(* Logix 5000 project; controller Amvex_Thorpe_Flowmeter vendor 1 type 14 code 106 rev 33.13; software revision 33.01; part 4 of 16 *)

ADD_ON_INSTRUCTION MoveLinRelTRF   (* revision 0.1, vendor Mecademic Inc., ExecuteEnableInFalse *)
// Relative movement (relative to the current TRF position)
VAR_IN_OUT
   RobotInputs : _061D:Meca500_86BDA20B:I:0; {required}
   RobotOutputs : _061D:Meca500_01F88326:O:0; {required}
END_VAR
VAR_INPUT
   Pose_X_Pos : REAL; {required}
   Pose_Y_Pos : REAL; {required}
   Pose_Z_Pos : REAL; {required}
   Pose_rX_Ang : REAL; {required}
   Pose_rY_Ang : REAL; {required}
   Pose_rZ_Ang : REAL; {required}
   ExternalStateControl : BOOL; {required}
   ExternalMoveID : INT; {required}
END_VAR
VAR_OUTPUT
   Enabled : BOOL; {visible}
   Sent : BOOL; {visible}
   Buffered : BOOL; {visible}
   Error : BOOL; {visible}
END_VAR
VAR
   InternalMoveID : INT; {access None}
   MoveIDTrig : BOOL; {access None}
   MoveIDUpdated : BOOL; {access None}
   OneShot : DINT; {access None}
   FirstScan : BOOL; {access None}
END_VAR

ROUTINE EnableInFalse   (* ladder *)
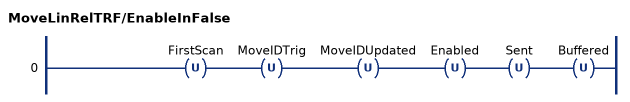
   0: OTU(FirstScan)OTU(MoveIDTrig)OTU(MoveIDUpdated)OTU(Enabled)OTU(Sent)OTU(Buffered);
END_ROUTINE

ROUTINE Logic   (* ladder *)
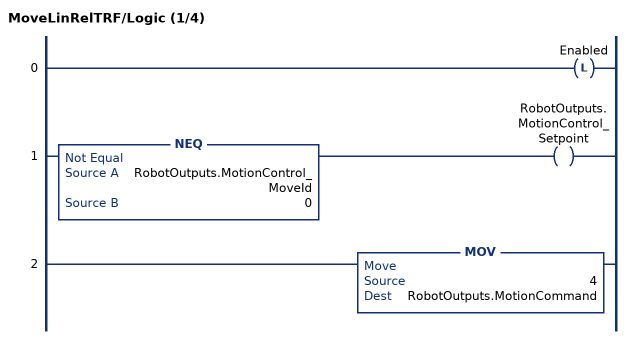
   0: OTL(Enabled);
   1: NEQ(RobotOutputs.MotionControl_MoveId,0)OTE(RobotOutputs.MotionControl_Setpoint);
   2: MOV(4,RobotOutputs.MotionCommand);
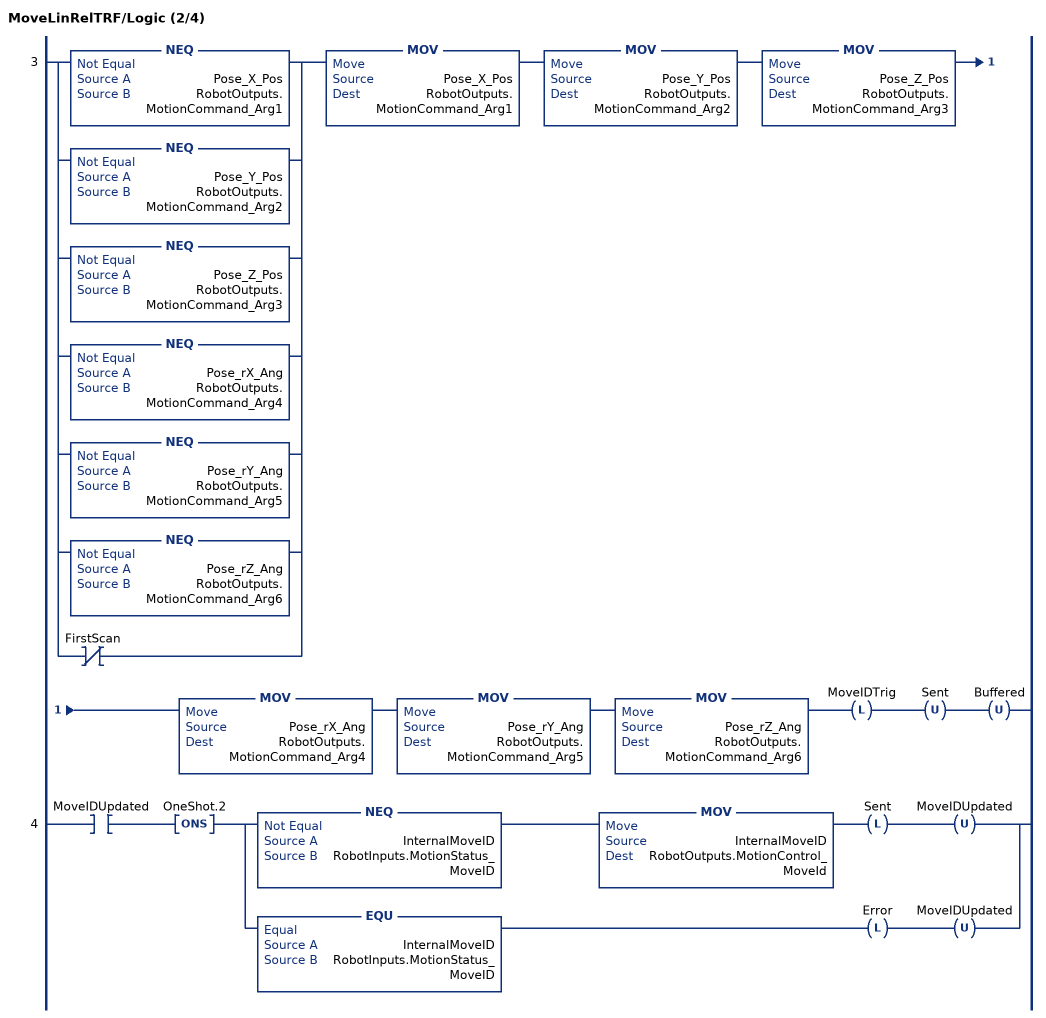
   3: [NEQ(Pose_X_Pos,RobotOutputs.MotionCommand_Arg1) ,NEQ(Pose_Y_Pos,RobotOutputs.MotionCommand_Arg2) ,NEQ(Pose_Z_Pos,RobotOutputs.MotionCommand_Arg3) ,NEQ(Pose_rX_Ang,RobotOutputs.MotionCommand_Arg4) ,NEQ(Pose_rY_Ang,RobotOutputs.MotionCommand_Arg5) ,NEQ(Pose_rZ_Ang,RobotOutputs.MotionCommand_Arg6) ,XIO(FirstScan) ]MOV(Pose_X_Pos,RobotOutputs.MotionCommand_Arg1)MOV(Pose_Y_Pos,RobotOutputs.MotionCommand_Arg2)MOV(Pose_Z_Pos,RobotOutputs.MotionCommand_Arg3)MOV(Pose_rX_Ang,RobotOutputs.MotionCommand_Arg4)MOV(Pose_rY_Ang,RobotOutputs.MotionCommand_Arg5)MOV(Pose_rZ_Ang,RobotOutputs.MotionCommand_Arg6)OTL(MoveIDTrig)OTU(Sent)OTU(Buffered);
   4: XIC(MoveIDUpdated)ONS(OneShot.2)[NEQ(InternalMoveID,RobotInputs.MotionStatus_MoveID) MOV(InternalMoveID,RobotOutputs.MotionControl_MoveId) OTL(Sent) OTU(MoveIDUpdated) ,EQU(InternalMoveID,RobotInputs.MotionStatus_MoveID) OTL(Error) OTU(MoveIDUpdated) ];
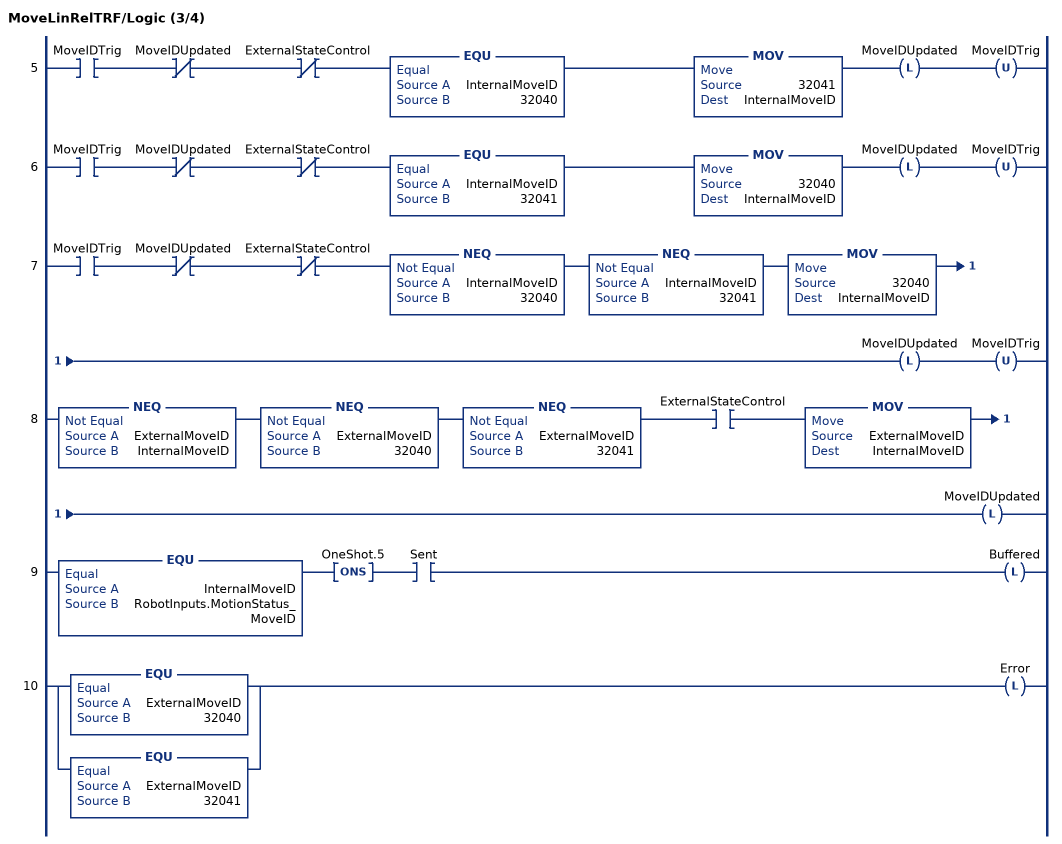
   5: XIC(MoveIDTrig)XIO(MoveIDUpdated)XIO(ExternalStateControl)EQU(InternalMoveID,32040)MOV(32041,InternalMoveID)OTL(MoveIDUpdated)OTU(MoveIDTrig);
   6: XIC(MoveIDTrig)XIO(MoveIDUpdated)XIO(ExternalStateControl)EQU(InternalMoveID,32041)MOV(32040,InternalMoveID)OTL(MoveIDUpdated)OTU(MoveIDTrig);
   7: XIC(MoveIDTrig)XIO(MoveIDUpdated)XIO(ExternalStateControl)NEQ(InternalMoveID,32040)NEQ(InternalMoveID,32041)MOV(32040,InternalMoveID)OTL(MoveIDUpdated)OTU(MoveIDTrig);
   8: NEQ(ExternalMoveID,InternalMoveID)NEQ(ExternalMoveID,32040)NEQ(ExternalMoveID,32041)XIC(ExternalStateControl)MOV(ExternalMoveID,InternalMoveID)OTL(MoveIDUpdated);
   9: EQU(InternalMoveID,RobotInputs.MotionStatus_MoveID)ONS(OneShot.5)XIC(Sent)OTL(Buffered);
   10: [EQU(ExternalMoveID,32040) ,EQU(ExternalMoveID,32041) ]OTL(Error);
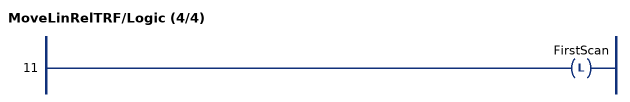
   11: OTL(FirstScan);
END_ROUTINE
END_ADD_ON_INSTRUCTION

ADD_ON_INSTRUCTION MoveLinRelWRF   (* revision 0.1, vendor Mecademic Inc., ExecuteEnableInFalse *)
// Relative movement (relative to the current WRF position)
VAR_IN_OUT
   RobotInputs : _061D:Meca500_86BDA20B:I:0; {required}
   RobotOutputs : _061D:Meca500_01F88326:O:0; {required}
END_VAR
VAR_INPUT
   Pose_X_Pos : REAL; {required}
   Pose_Y_Pos : REAL; {required}
   Pose_Z_Pos : REAL; {required}
   Pose_rX_Ang : REAL; {required}
   Pose_rY_Ang : REAL; {required}
   Pose_rZ_Ang : REAL; {required}
   ExternalStateControl : BOOL; {required}
   ExternalMoveID : INT; {required}
END_VAR
VAR_OUTPUT
   Enabled : BOOL; {visible}
   Sent : BOOL; {visible}
   Buffered : BOOL; {visible}
   Error : BOOL; {visible}
END_VAR
VAR
   InternalMoveID : INT; {access None}
   MoveIDTrig : BOOL; {access None}
   MoveIDUpdated : BOOL; {access None}
   OneShot : DINT; {access None}
   FirstScan : BOOL; {access None}
END_VAR

ROUTINE EnableInFalse   (* ladder *)
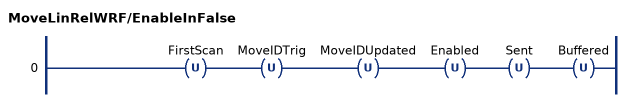
   0: OTU(FirstScan)OTU(MoveIDTrig)OTU(MoveIDUpdated)OTU(Enabled)OTU(Sent)OTU(Buffered);
END_ROUTINE

ROUTINE Logic   (* ladder *)
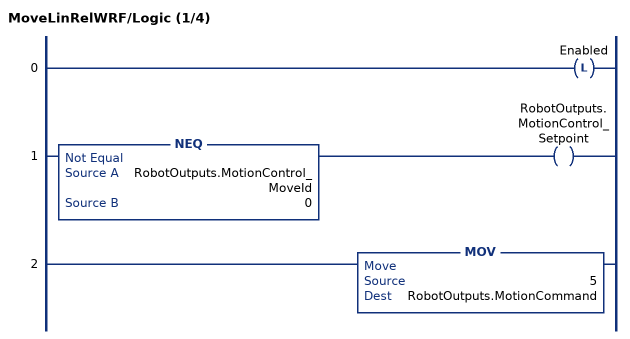
   0: OTL(Enabled);
   1: NEQ(RobotOutputs.MotionControl_MoveId,0)OTE(RobotOutputs.MotionControl_Setpoint);
   2: MOV(5,RobotOutputs.MotionCommand);
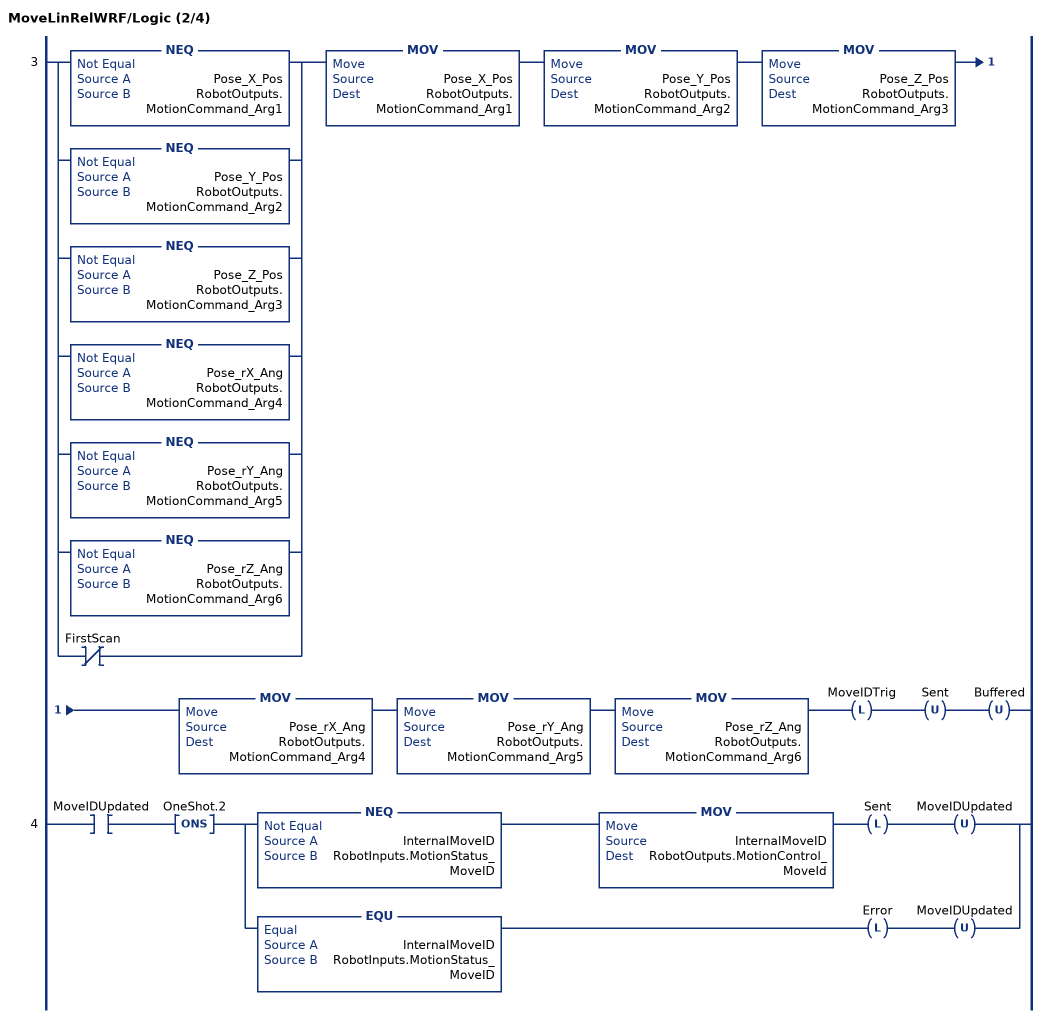
   3: [NEQ(Pose_X_Pos,RobotOutputs.MotionCommand_Arg1) ,NEQ(Pose_Y_Pos,RobotOutputs.MotionCommand_Arg2) ,NEQ(Pose_Z_Pos,RobotOutputs.MotionCommand_Arg3) ,NEQ(Pose_rX_Ang,RobotOutputs.MotionCommand_Arg4) ,NEQ(Pose_rY_Ang,RobotOutputs.MotionCommand_Arg5) ,NEQ(Pose_rZ_Ang,RobotOutputs.MotionCommand_Arg6) ,XIO(FirstScan) ]MOV(Pose_X_Pos,RobotOutputs.MotionCommand_Arg1)MOV(Pose_Y_Pos,RobotOutputs.MotionCommand_Arg2)MOV(Pose_Z_Pos,RobotOutputs.MotionCommand_Arg3)MOV(Pose_rX_Ang,RobotOutputs.MotionCommand_Arg4)MOV(Pose_rY_Ang,RobotOutputs.MotionCommand_Arg5)MOV(Pose_rZ_Ang,RobotOutputs.MotionCommand_Arg6)OTL(MoveIDTrig)OTU(Sent)OTU(Buffered);
   4: XIC(MoveIDUpdated)ONS(OneShot.2)[NEQ(InternalMoveID,RobotInputs.MotionStatus_MoveID) MOV(InternalMoveID,RobotOutputs.MotionControl_MoveId) OTL(Sent) OTU(MoveIDUpdated) ,EQU(InternalMoveID,RobotInputs.MotionStatus_MoveID) OTL(Error) OTU(MoveIDUpdated) ];
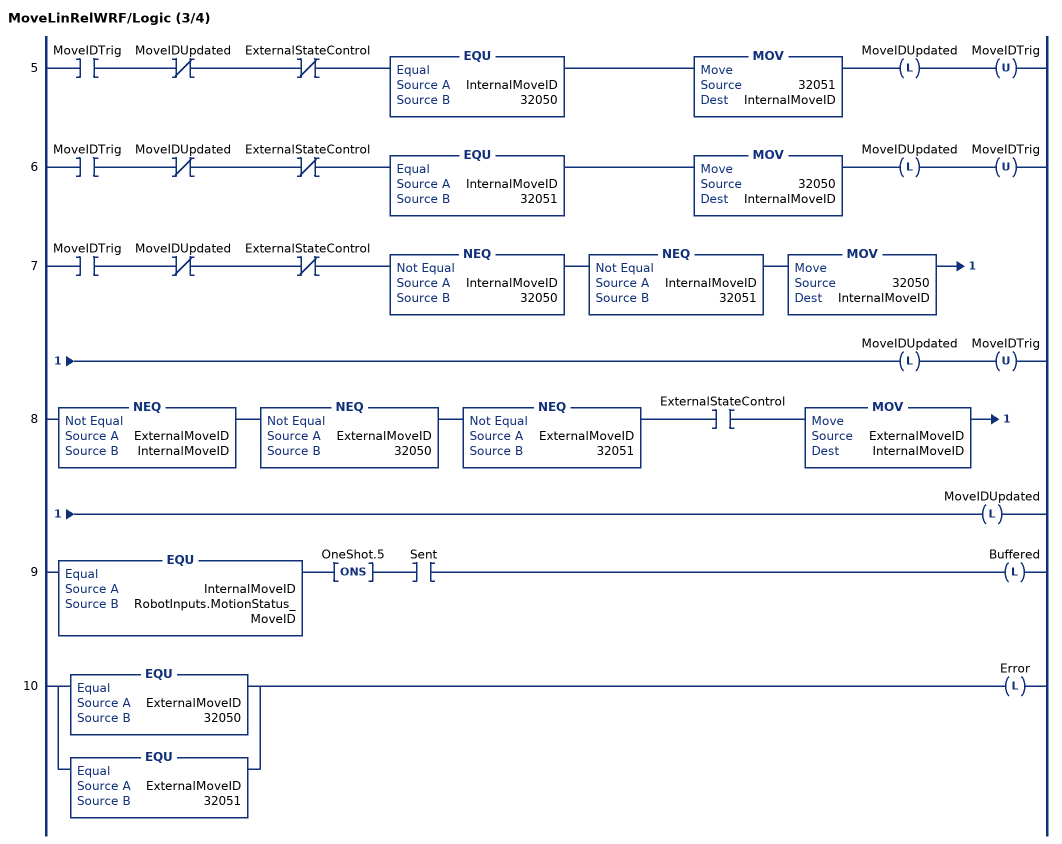
   5: XIC(MoveIDTrig)XIO(MoveIDUpdated)XIO(ExternalStateControl)EQU(InternalMoveID,32050)MOV(32051,InternalMoveID)OTL(MoveIDUpdated)OTU(MoveIDTrig);
   6: XIC(MoveIDTrig)XIO(MoveIDUpdated)XIO(ExternalStateControl)EQU(InternalMoveID,32051)MOV(32050,InternalMoveID)OTL(MoveIDUpdated)OTU(MoveIDTrig);
   7: XIC(MoveIDTrig)XIO(MoveIDUpdated)XIO(ExternalStateControl)NEQ(InternalMoveID,32050)NEQ(InternalMoveID,32051)MOV(32050,InternalMoveID)OTL(MoveIDUpdated)OTU(MoveIDTrig);
   8: NEQ(ExternalMoveID,InternalMoveID)NEQ(ExternalMoveID,32050)NEQ(ExternalMoveID,32051)XIC(ExternalStateControl)MOV(ExternalMoveID,InternalMoveID)OTL(MoveIDUpdated);
   9: EQU(InternalMoveID,RobotInputs.MotionStatus_MoveID)ONS(OneShot.5)XIC(Sent)OTL(Buffered);
   10: [EQU(ExternalMoveID,32050) ,EQU(ExternalMoveID,32051) ]OTL(Error);
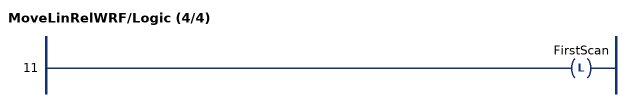
   11: OTL(FirstScan);
END_ROUTINE
END_ADD_ON_INSTRUCTION

ADD_ON_INSTRUCTION MoveLinVelTRF   (* revision 0.1, vendor Mecademic Inc., ExecuteEnableInFalse *)
// Set current mode to "cartesian TRF velocity mode"
VAR_IN_OUT
   RobotInputs : _061D:Meca500_86BDA20B:I:0; {required}
   RobotOutputs : _061D:Meca500_01F88326:O:0; {required}
END_VAR
VAR_INPUT
   Pose_X_Vel : REAL; {required}
   Pose_Y_Vel : REAL; {required}
   Pose_Z_Vel : REAL; {required}
   Pose_rX_Vel : REAL; {required}
   Pose_rY_Vel : REAL; {required}
   Pose_rZ_Vel : REAL; {required}
   ExternalStateControl : BOOL; {required}
   ExternalMoveID : INT; {required}
END_VAR
VAR_OUTPUT
   Enabled : BOOL; {visible}
   Sent : BOOL; {visible}
   Buffered : BOOL; {visible}
   Error : BOOL; {visible}
END_VAR
VAR
   InternalMoveID : INT; {access None}
   MoveIDTrig : BOOL; {access None}
   MoveIDUpdated : BOOL; {access None}
   OneShot : DINT; {access None}
   FirstScan : BOOL; {access None}
END_VAR

ROUTINE EnableInFalse   (* ladder *)
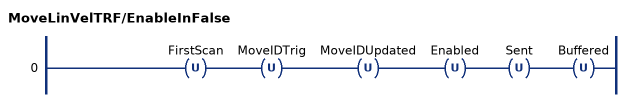
   0: OTU(FirstScan)OTU(MoveIDTrig)OTU(MoveIDUpdated)OTU(Enabled)OTU(Sent)OTU(Buffered);
END_ROUTINE

ROUTINE Logic   (* ladder *)
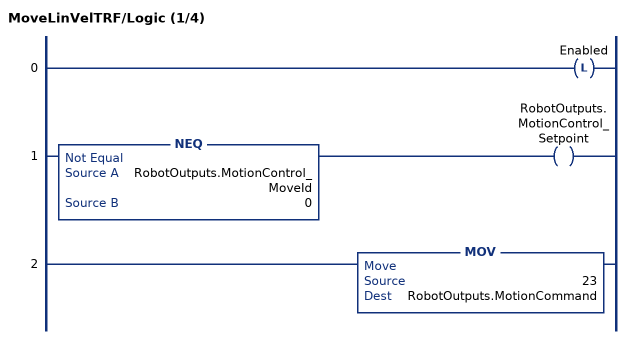
   0: OTL(Enabled);
   1: NEQ(RobotOutputs.MotionControl_MoveId,0)OTE(RobotOutputs.MotionControl_Setpoint);
   2: MOV(23,RobotOutputs.MotionCommand);
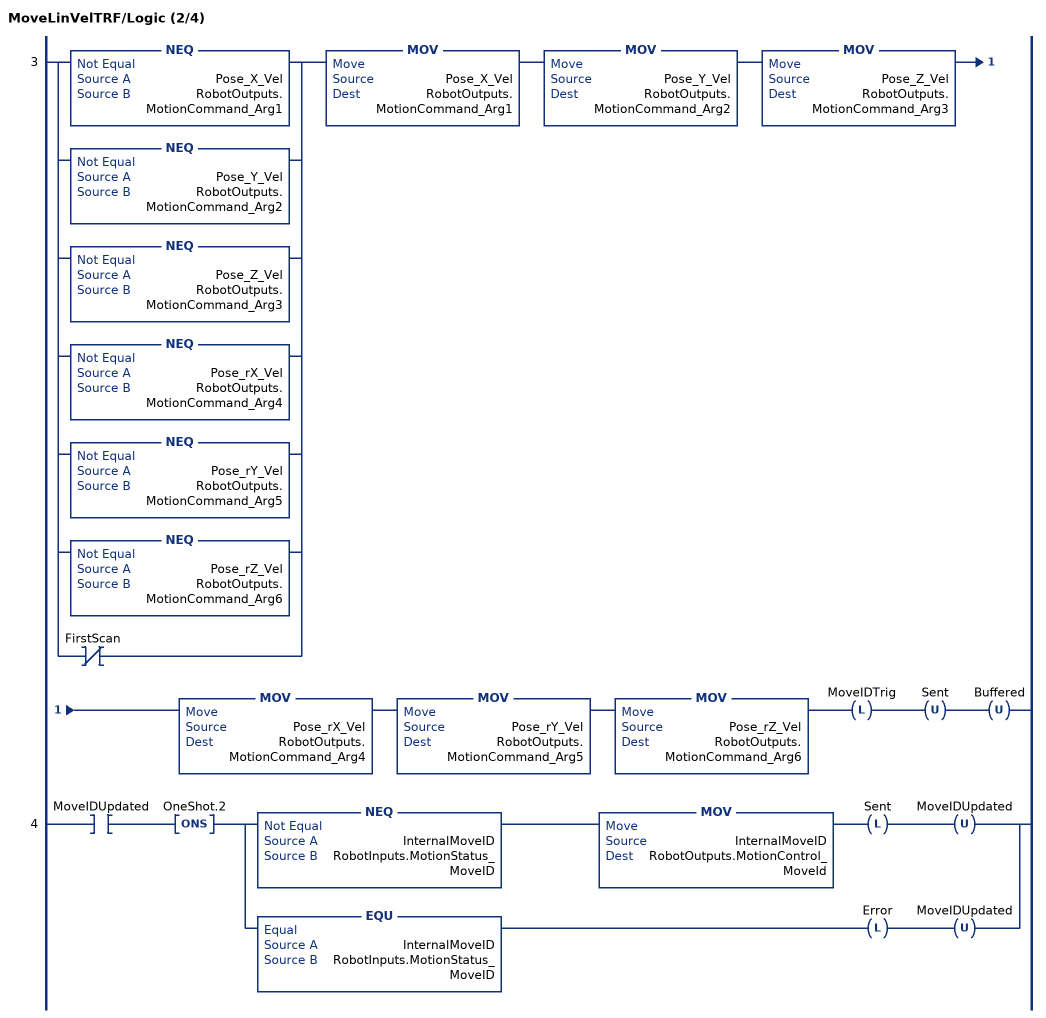
   3: [NEQ(Pose_X_Vel,RobotOutputs.MotionCommand_Arg1) ,NEQ(Pose_Y_Vel,RobotOutputs.MotionCommand_Arg2) ,NEQ(Pose_Z_Vel,RobotOutputs.MotionCommand_Arg3) ,NEQ(Pose_rX_Vel,RobotOutputs.MotionCommand_Arg4) ,NEQ(Pose_rY_Vel,RobotOutputs.MotionCommand_Arg5) ,NEQ(Pose_rZ_Vel,RobotOutputs.MotionCommand_Arg6) ,XIO(FirstScan) ]MOV(Pose_X_Vel,RobotOutputs.MotionCommand_Arg1)MOV(Pose_Y_Vel,RobotOutputs.MotionCommand_Arg2)MOV(Pose_Z_Vel,RobotOutputs.MotionCommand_Arg3)MOV(Pose_rX_Vel,RobotOutputs.MotionCommand_Arg4)MOV(Pose_rY_Vel,RobotOutputs.MotionCommand_Arg5)MOV(Pose_rZ_Vel,RobotOutputs.MotionCommand_Arg6)OTL(MoveIDTrig)OTU(Sent)OTU(Buffered);
   4: XIC(MoveIDUpdated)ONS(OneShot.2)[NEQ(InternalMoveID,RobotInputs.MotionStatus_MoveID) MOV(InternalMoveID,RobotOutputs.MotionControl_MoveId) OTL(Sent) OTU(MoveIDUpdated) ,EQU(InternalMoveID,RobotInputs.MotionStatus_MoveID) OTL(Error) OTU(MoveIDUpdated) ];
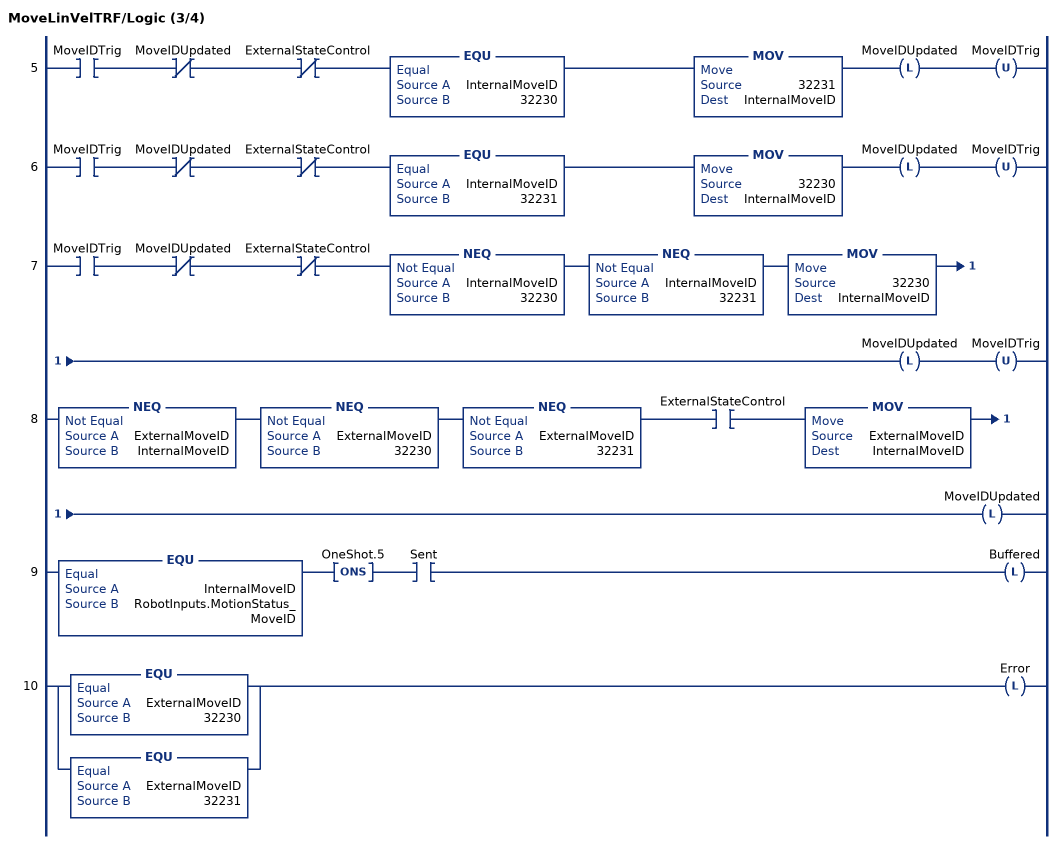
   5: XIC(MoveIDTrig)XIO(MoveIDUpdated)XIO(ExternalStateControl)EQU(InternalMoveID,32230)MOV(32231,InternalMoveID)OTL(MoveIDUpdated)OTU(MoveIDTrig);
   6: XIC(MoveIDTrig)XIO(MoveIDUpdated)XIO(ExternalStateControl)EQU(InternalMoveID,32231)MOV(32230,InternalMoveID)OTL(MoveIDUpdated)OTU(MoveIDTrig);
   7: XIC(MoveIDTrig)XIO(MoveIDUpdated)XIO(ExternalStateControl)NEQ(InternalMoveID,32230)NEQ(InternalMoveID,32231)MOV(32230,InternalMoveID)OTL(MoveIDUpdated)OTU(MoveIDTrig);
   8: NEQ(ExternalMoveID,InternalMoveID)NEQ(ExternalMoveID,32230)NEQ(ExternalMoveID,32231)XIC(ExternalStateControl)MOV(ExternalMoveID,InternalMoveID)OTL(MoveIDUpdated);
   9: EQU(InternalMoveID,RobotInputs.MotionStatus_MoveID)ONS(OneShot.5)XIC(Sent)OTL(Buffered);
   10: [EQU(ExternalMoveID,32230) ,EQU(ExternalMoveID,32231) ]OTL(Error);
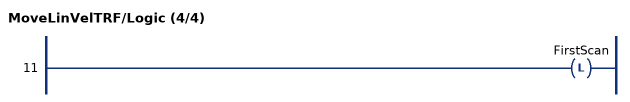
   11: OTL(FirstScan);
END_ROUTINE
END_ADD_ON_INSTRUCTION

ADD_ON_INSTRUCTION MoveLinVelWRF   (* revision 0.1, vendor Mecademic Inc., ExecuteEnableInFalse *)
// Set current mode to "cartesian WRF velocity mode"
VAR_IN_OUT
   RobotInputs : _061D:Meca500_86BDA20B:I:0; {required}
   RobotOutputs : _061D:Meca500_01F88326:O:0; {required}
END_VAR
VAR_INPUT
   Pose_X_Vel : REAL; {required}
   Pose_Y_Vel : REAL; {required}
   Pose_Z_Vel : REAL; {required}
   Pose_rX_Vel : REAL; {required}
   Pose_rY_Vel : REAL; {required}
   Pose_rZ_Vel : REAL; {required}
   ExternalStateControl : BOOL; {required}
   ExternalMoveID : INT; {required}
END_VAR
VAR_OUTPUT
   Enabled : BOOL; {visible}
   Sent : BOOL; {visible}
   Buffered : BOOL; {visible}
   Error : BOOL; {visible}
END_VAR
VAR
   InternalMoveID : INT; {access None}
   MoveIDTrig : BOOL; {access None}
   MoveIDUpdated : BOOL; {access None}
   OneShot : DINT; {access None}
   FirstScan : BOOL; {access None}
END_VAR

ROUTINE EnableInFalse   (* ladder *)
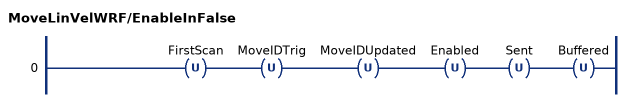
   0: OTU(FirstScan)OTU(MoveIDTrig)OTU(MoveIDUpdated)OTU(Enabled)OTU(Sent)OTU(Buffered);
END_ROUTINE

ROUTINE Logic   (* ladder *)
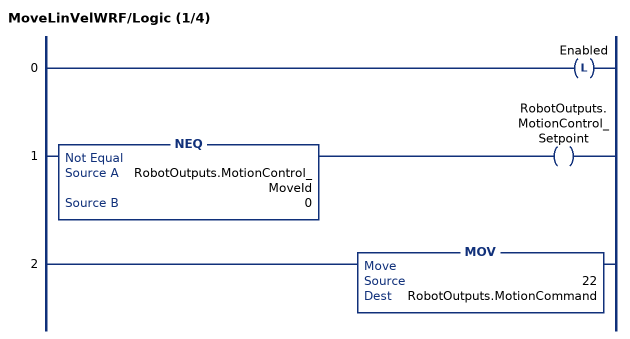
   0: OTL(Enabled);
   1: NEQ(RobotOutputs.MotionControl_MoveId,0)OTE(RobotOutputs.MotionControl_Setpoint);
   2: MOV(22,RobotOutputs.MotionCommand);
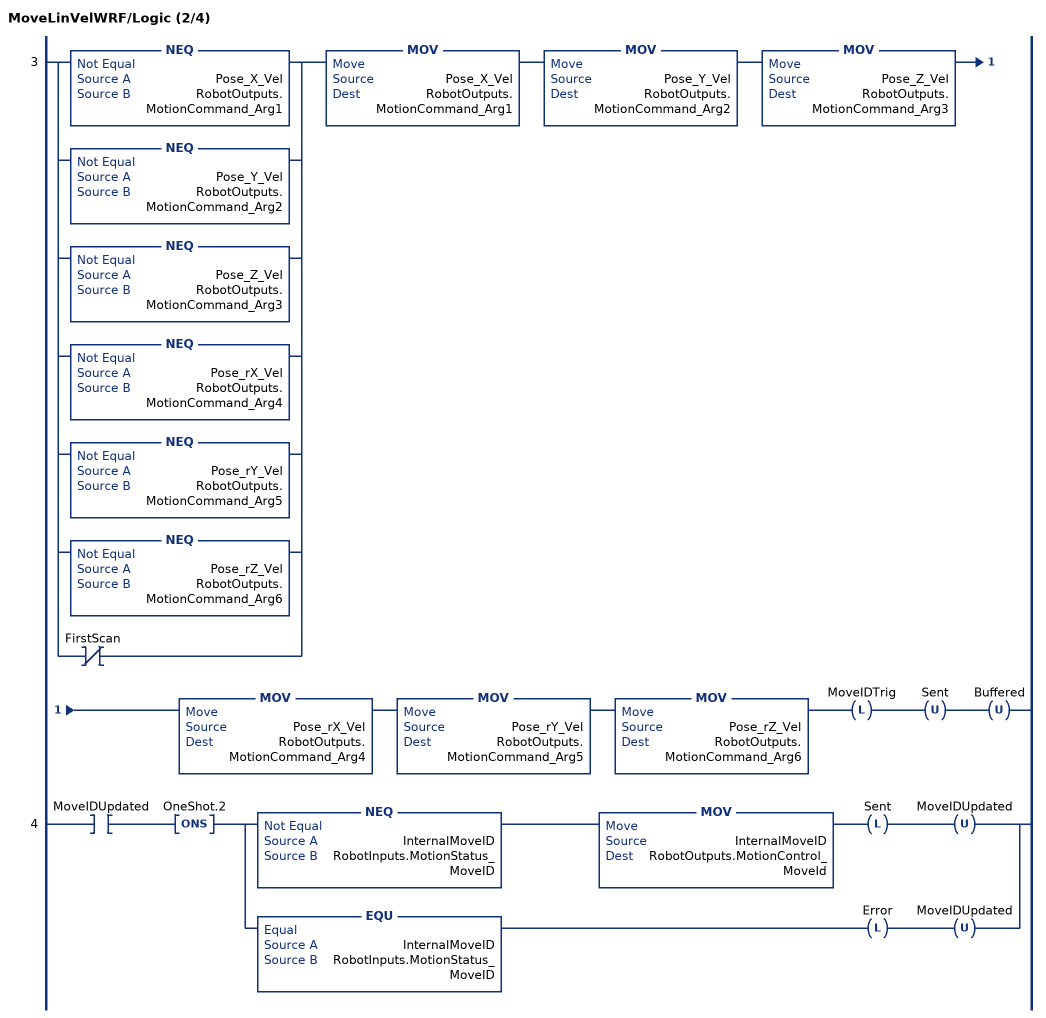
   3: [NEQ(Pose_X_Vel,RobotOutputs.MotionCommand_Arg1) ,NEQ(Pose_Y_Vel,RobotOutputs.MotionCommand_Arg2) ,NEQ(Pose_Z_Vel,RobotOutputs.MotionCommand_Arg3) ,NEQ(Pose_rX_Vel,RobotOutputs.MotionCommand_Arg4) ,NEQ(Pose_rY_Vel,RobotOutputs.MotionCommand_Arg5) ,NEQ(Pose_rZ_Vel,RobotOutputs.MotionCommand_Arg6) ,XIO(FirstScan) ]MOV(Pose_X_Vel,RobotOutputs.MotionCommand_Arg1)MOV(Pose_Y_Vel,RobotOutputs.MotionCommand_Arg2)MOV(Pose_Z_Vel,RobotOutputs.MotionCommand_Arg3)MOV(Pose_rX_Vel,RobotOutputs.MotionCommand_Arg4)MOV(Pose_rY_Vel,RobotOutputs.MotionCommand_Arg5)MOV(Pose_rZ_Vel,RobotOutputs.MotionCommand_Arg6)OTL(MoveIDTrig)OTU(Sent)OTU(Buffered);
   4: XIC(MoveIDUpdated)ONS(OneShot.2)[NEQ(InternalMoveID,RobotInputs.MotionStatus_MoveID) MOV(InternalMoveID,RobotOutputs.MotionControl_MoveId) OTL(Sent) OTU(MoveIDUpdated) ,EQU(InternalMoveID,RobotInputs.MotionStatus_MoveID) OTL(Error) OTU(MoveIDUpdated) ];
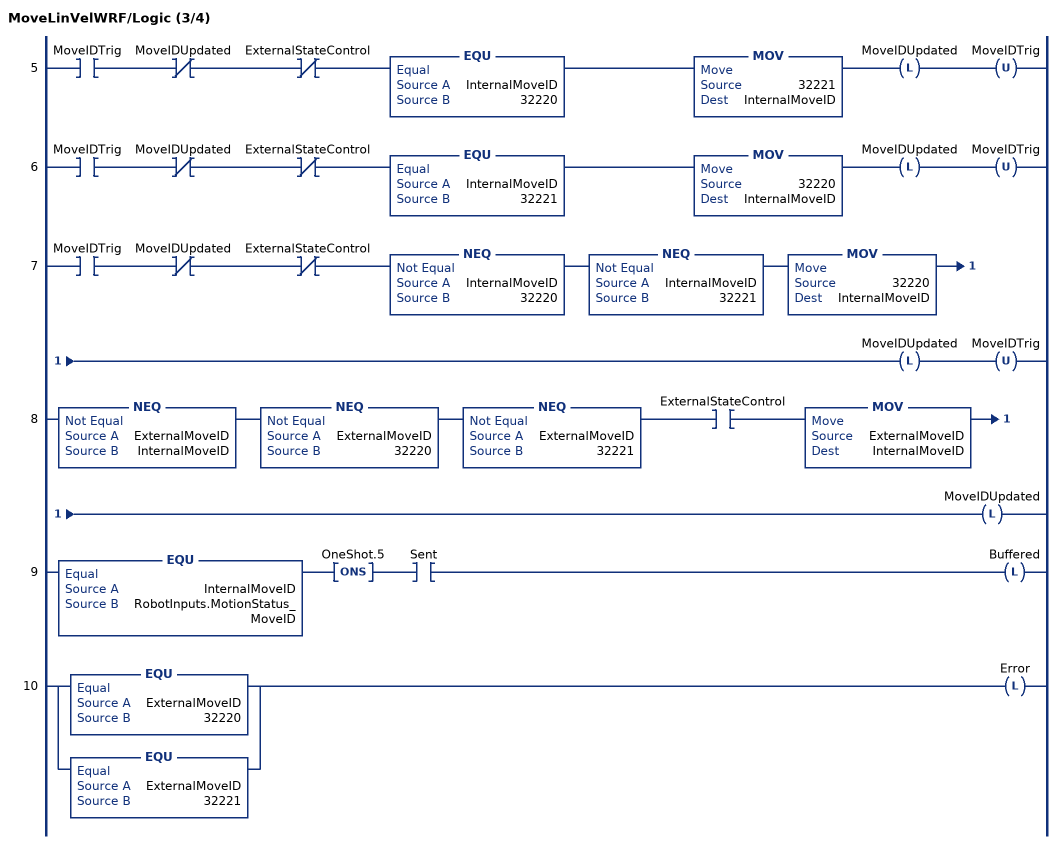
   5: XIC(MoveIDTrig)XIO(MoveIDUpdated)XIO(ExternalStateControl)EQU(InternalMoveID,32220)MOV(32221,InternalMoveID)OTL(MoveIDUpdated)OTU(MoveIDTrig);
   6: XIC(MoveIDTrig)XIO(MoveIDUpdated)XIO(ExternalStateControl)EQU(InternalMoveID,32221)MOV(32220,InternalMoveID)OTL(MoveIDUpdated)OTU(MoveIDTrig);
   7: XIC(MoveIDTrig)XIO(MoveIDUpdated)XIO(ExternalStateControl)NEQ(InternalMoveID,32220)NEQ(InternalMoveID,32221)MOV(32220,InternalMoveID)OTL(MoveIDUpdated)OTU(MoveIDTrig);
   8: NEQ(ExternalMoveID,InternalMoveID)NEQ(ExternalMoveID,32220)NEQ(ExternalMoveID,32221)XIC(ExternalStateControl)MOV(ExternalMoveID,InternalMoveID)OTL(MoveIDUpdated);
   9: EQU(InternalMoveID,RobotInputs.MotionStatus_MoveID)ONS(OneShot.5)XIC(Sent)OTL(Buffered);
   10: [EQU(ExternalMoveID,32220) ,EQU(ExternalMoveID,32221) ]OTL(Error);
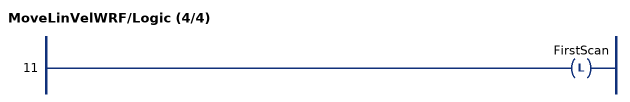
   11: OTL(FirstScan);
END_ROUTINE
END_ADD_ON_INSTRUCTION
